# EPICS StreamDevice protocol: dn1-epics/dn1App/Db/simple.proto
Terminator = CR LF;
getval {
 in "%d";
}
